// TIA Portal V16 program export: 1 tag tables, 0 data types, 0 data blocks, 6 code blocks (in call order from the OBs), 0 instance data blocks

VAR_GLOBAL   // PLC tag table "Standard-Variablentabelle"
   "Auto/Manual" AT %I0.0 : Bool;
   Start AT %I0.1 : Bool;
   Reset AT %I0.2 : Bool;
   Stop AT %I0.3 : Bool;
   Estop AT %I0.4 : Bool;
   "Conveyor Sensor 1" AT %I0.5 : Bool;
   "Conveyor Sensor 2" AT %I0.6 : Bool;
   "Conveyor Sensor 3" AT %I0.7 : Bool;
   "Alarm Siren" AT %Q0.0 : Bool;
   "Start Light" AT %Q0.1 : Bool;
   "Reset Light" AT %Q0.2 : Bool;
   "Stop Light" AT %Q0.3 : Bool;
   "Pusher 2" AT %Q0.5 : Bool;
   "Stack Light Green" AT %Q0.6 : Bool;
   "Stack Light Yellow" AT %Q0.7 : Bool;
   "Ready to Run" AT %M0.0 : Bool;
   "Reset Memory" AT %M0.5 : Bool;
   "Pusher Sensor 1 Mem" AT %M0.6 : Bool;
   "Pusher 1 FW Mem" AT %M0.7 : Bool;
   "Pusher Sensor 2 Mem" AT %M1.0 : Bool;
   "Pusher 2 FW Mem" AT %M1.1 : Bool;
   "Conveyor Sensor 4" AT %I1.0 : Bool;
   "Pusher Sensor 1" AT %I1.1 : Bool;
   "Pusher Sensor 2" AT %I1.2 : Bool;
   "Pusher 1 FW" AT %I1.3 : Bool;
   "Pusher 2 FW" AT %I1.4 : Bool;
   "Pusher 1" AT %Q0.4 : Bool;
   "Stack Light Red" AT %Q1.0 : Bool;
   "Drain 1" AT %Q1.1 : Bool;
   "Drain 2" AT %Q1.2 : Bool;
   "Drain 3" AT %Q1.3 : Bool;
   "Conveyor 1" AT %QW36 : Int;
   "Conveyor 2" AT %Q1.5 : Bool;
   "Conveyor 3" AT %Q1.6 : Bool;
   "Conveyor 4" AT %Q1.7 : Bool;
   "Conveyor Sensor 1 Mem" AT %M1.2 : Bool;
   "Conveyor Sensor 2 Mem" AT %M1.3 : Bool;
   "Conveyor Sensor 3 Mem" AT %M1.4 : Bool;
   "Conveyor Sensor 4 Mem" AT %M1.5 : Bool;
   "Conveyor Sensor 5 Mem" AT %M1.6 : Bool;
   "Advanced Feeder" AT %Q2.1 : Bool;
   "Conveyor Sensor 5" AT %I1.5 : Bool;
   "Running Torque" AT %IW30 : Int;
   "Running Temperature" AT %IW32 : Int;
   "Error Message" AT %Q2.2 : Bool;
   "1.5 KG" AT %QW30 : Int;
   "5.0 KG" AT %QW32 : Int;
   "7.5" AT %QW34 : Int;
   "Estop Memory" AT %M0.1 : Bool;
END_VAR

ORGANIZATION_BLOCK "Main"   // OB1, LAD, ProgramCycle
TITLE = "Main Program Sweep (Cycle)"
{ S7_Optimized_Access := 'TRUE' }
VERSION : 0.1
// stored: AutoNumber true, IsIECCheckEnabled false, SetENOAutomatically false
   VAR_INPUT
      Initial_Call : Bool;   // Initial call of this OB
      Remanence : Bool;   // =True, if remanent data are available
   END_VAR
BEGIN

REGION Network 1
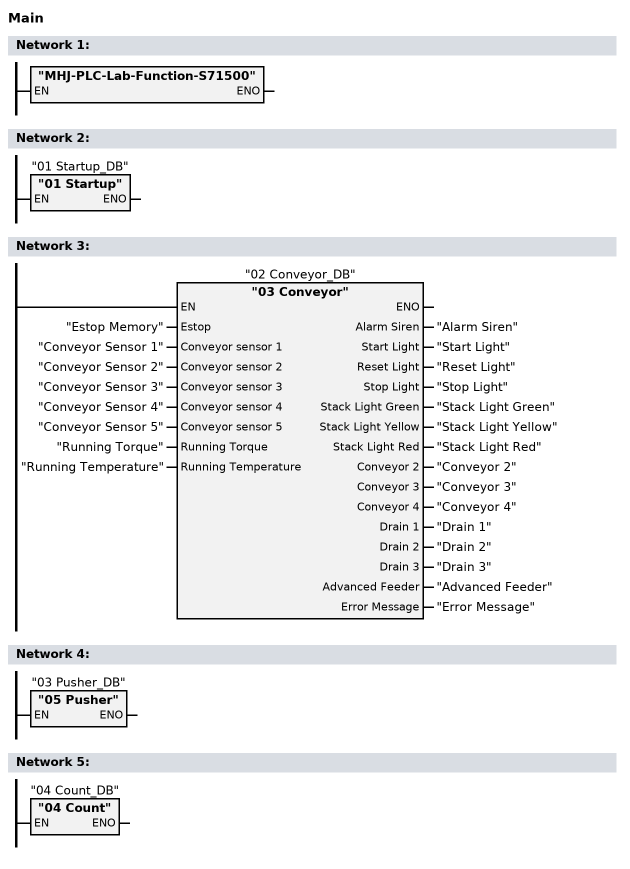
   RUNG wire#powerrail
      "MHJ-PLC-Lab-Function-S71500"()
   END_RUNG
   // the same network as SCL:
   "MHJ-PLC-Lab-Function-S71500"();
END_REGION

REGION Network 2
   RUNG wire#powerrail
      "01 Startup_DB"()
   END_RUNG
   // the same network as SCL:
   "01 Startup_DB"();   // "01 Startup"
END_REGION

REGION Network 3
   RUNG wire#powerrail
      "02 Conveyor_DB"(Estop := "Estop Memory", "Conveyor sensor 1" := "Conveyor Sensor 1", "Conveyor sensor 2" := "Conveyor Sensor 2", "Conveyor sensor 3" := "Conveyor Sensor 3", "Conveyor sensor 4" := "Conveyor Sensor 4", "Conveyor sensor 5" := "Conveyor Sensor 5", "Running Torque" := "Running Torque", "Running Temperature" := "Running Temperature", "Alarm Siren" => "Alarm Siren", "Start Light" => "Start Light", "Reset Light" => "Reset Light", "Stop Light" => "Stop Light", "Stack Light Green" => "Stack Light Green", "Stack Light Yellow" => "Stack Light Yellow", "Stack Light Red" => "Stack Light Red", "Conveyor 2" => "Conveyor 2", "Conveyor 3" => "Conveyor 3", "Conveyor 4" => "Conveyor 4", "Drain 1" => "Drain 1", "Drain 2" => "Drain 2", "Drain 3" => "Drain 3", "Advanced Feeder" => "Advanced Feeder", "Error Message" => "Error Message")
   END_RUNG
   // the same network as SCL:
   "02 Conveyor_DB"(Estop := "Estop Memory",   // "03 Conveyor"
                    "Conveyor sensor 1" := "Conveyor Sensor 1",
                    "Conveyor sensor 2" := "Conveyor Sensor 2",
                    "Conveyor sensor 3" := "Conveyor Sensor 3",
                    "Conveyor sensor 4" := "Conveyor Sensor 4",
                    "Conveyor sensor 5" := "Conveyor Sensor 5",
                    "Running Torque" := "Running Torque",
                    "Running Temperature" := "Running Temperature",
                    "Alarm Siren" => "Alarm Siren",
                    "Start Light" => "Start Light",
                    "Reset Light" => "Reset Light",
                    "Stop Light" => "Stop Light",
                    "Stack Light Green" => "Stack Light Green",
                    "Stack Light Yellow" => "Stack Light Yellow",
                    "Stack Light Red" => "Stack Light Red",
                    "Conveyor 2" => "Conveyor 2",
                    "Conveyor 3" => "Conveyor 3",
                    "Conveyor 4" => "Conveyor 4",
                    "Drain 1" => "Drain 1",
                    "Drain 2" => "Drain 2",
                    "Drain 3" => "Drain 3",
                    "Advanced Feeder" => "Advanced Feeder",
                    "Error Message" => "Error Message");
END_REGION

REGION Network 4
   RUNG wire#powerrail
      "03 Pusher_DB"()
   END_RUNG
   // the same network as SCL:
   "03 Pusher_DB"();   // "05 Pusher"
END_REGION

REGION Network 5
   RUNG wire#powerrail
      "04 Count_DB"()
   END_RUNG
   // the same network as SCL:
   "04 Count_DB"();   // "04 Count"
END_REGION
END_ORGANIZATION_BLOCK

FUNCTION_BLOCK "01 Startup"   // FB1, LAD
{ S7_Optimized_Access := 'TRUE' }
VERSION : 0.1
// stored: AutoNumber true, IsIECCheckEnabled false, IsRetainMemResEnabled false, MemoryReserve 100, SetENOAutomatically false, UDAEnableTagReadback false
   VAR_TEMP   // added for the SCL form of the ladder/FBD networks
      _w1 : Bool;
   END_VAR
BEGIN

REGION Network 1: Run Mode
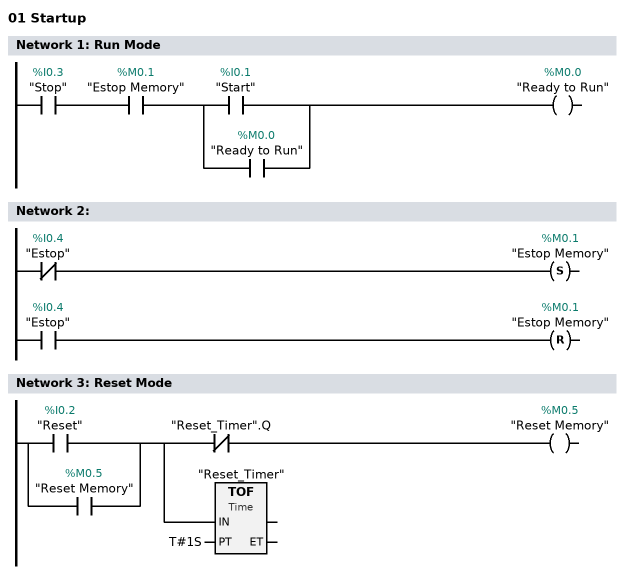
   RUNG wire#powerrail
      Contact( "Stop" )
      Contact( "Estop Memory" )
      wire#w1
      Contact( "Start" )
      wire#w2
      Coil( "Ready to Run" )
   END_RUNG
   RUNG wire#w1
      Contact( "Ready to Run" )
   END_RUNG wire#w2
   // the same network as SCL:
   "Ready to Run" := "Stop" AND "Estop Memory" AND ("Start" OR "Ready to Run");
END_REGION

REGION Network 2
   RUNG wire#powerrail
      I_Contact( "Estop" )
      S_Coil( "Estop Memory" )
   END_RUNG
   RUNG wire#powerrail
      Contact( "Estop" )
      R_Coil( "Estop Memory" )
   END_RUNG
   // the same network as SCL:
   IF NOT "Estop" THEN "Estop Memory" := TRUE; END_IF;
   IF "Estop" THEN "Estop Memory" := FALSE; END_IF;
END_REGION

REGION Network 3: Reset Mode
   RUNG wire#powerrail
      Contact( "Reset" )
      wire#w1
      I_Contact( "Reset_Timer".Q )
      Coil( "Reset Memory" )
   END_RUNG
   RUNG wire#powerrail
      Contact( "Reset Memory" )
   END_RUNG wire#w1
   RUNG wire#w1
      { S7_Templates := "time_type := Time" } "Reset_Timer".TOF(pt := T#1S, et =>)
   END_RUNG
   // the same network as SCL:
   #_w1 := "Reset" OR "Reset Memory";
   "Reset Memory" := #_w1 AND NOT "Reset_Timer".Q;
   "Reset_Timer".TOF(IN := #_w1, PT := T#1S);
END_REGION
END_FUNCTION_BLOCK

FUNCTION_BLOCK "03 Conveyor"
{ S7_Optimized_Access := 'TRUE' }
VERSION : 0.1
   VAR_INPUT 
      Estop : Bool;
      "Conveyor sensor 1" : Bool;
      "Conveyor sensor 2" : Bool;
      "Conveyor sensor 3" : Bool;
      "Conveyor sensor 4" : Bool;
      "Conveyor sensor 5" : Bool;
      "Running Torque" : Int;
      "Running Temperature" : Int;
   END_VAR

   VAR_OUTPUT 
      "Alarm Siren" : Bool;
      "Start Light" : Bool;
      "Reset Light" : Bool;
      "Stop Light" : Bool;
      "Stack Light Green" : Bool;
      "Stack Light Yellow" : Bool;
      "Stack Light Red" : Bool;
      "Conveyor 2" : Bool;
      "Conveyor 3" : Bool;
      "Conveyor 4" : Bool;
      "Drain 1" : Bool;
      "Drain 2" : Bool;
      "Drain 3" : Bool;
      "Advanced Feeder" : Bool;
      "Error Message" : Bool;
   END_VAR

   VAR 
      ET : Time;
      Error : Bool;
   END_VAR


BEGIN
	
	REGION Supply
	    IF "Ready to Run" THEN
	        // Statement section IF
	        #"Advanced Feeder" := TRUE;
	    END_IF;
	    
	    //CONVEYOR 2-5 CONTROL
	    
	    //Conveyor 2
	    IF "Ready to Run" THEN
	        IF #"Conveyor sensor 2" THEN
	            #"Conveyor 2" := TRUE;
	
	            "TOF_2".TOF (IN := #"Conveyor sensor 2",
	            PT := T#30s,
	            Q => #"Conveyor 2",
	            ET => #ET);
	        END_IF
	        ;
	    END_IF;
	    
	    IF "Ready to Run" THEN
	        IF #"Conveyor sensor 3" THEN
	            #"Conveyor 3" := TRUE;
	            
	            "TOF_3".TOF (IN := #"Conveyor sensor 3",
	            PT := T#30s,
	            Q => #"Conveyor 3",
	            ET => #ET);
	            
	        END_IF
	        ;
	    END_IF;
	    
	    IF "Ready to Run" THEN
	        IF #"Conveyor sensor 4" THEN
	            #"Conveyor 4" := TRUE;
	            
	            "TOF_4".TOF (IN := #"Conveyor sensor 4",
	            PT := T#30s,
	            Q => #"Conveyor 4",
	            ET => #ET);
	            
	        END_IF
	        ;
	    END_IF;
	    
	           
	END_REGION
	
	
	REGION Predictive Maintenace
	    
	    IF "Ready to Run" THEN
	        // Statement section IF
	        
	        // IF #"Running Torq > #"Rated Torque"OR #"Running Temperature"> #"Rated Temperature" THEN
	        IF #"Running Torque" > 6 OR #"Running Temperature" > 30 THEN
	            #"Error Message" := TRUE;
	            
	            "Timer_Error".TOF (IN := "Ready to Run",
	            PT := T#300s,
	            Q => #"Error Message",
	            ET => #ET);
	        END_IF;
	    END_IF;
	    
	    IF "Ready to Run" THEN
	        // Statement section IF
	        
	        // IF #"Running Torq > #"Rated Torque"OR #"Running Temperature"> #"Rated Temperature" THEN
	        IF #"Running Torque" > 6 OR #"Running Temperature" > 30 THEN
	            #"Estop" := TRUE;
	            
	            "Timer_Error".TOF(IN := "Ready to Run",
	                              PT := T#600s,
	                              Q => #"Error Message",
	                              ET => #ET);
	        END_IF;
	    END_IF;
	    
	END_REGION
	REGION End
	    IF "Ready to Run" THEN
	        #"Drain 1" := TRUE;
	        #"Drain 2" := TRUE;
	        #"Drain 3" := TRUE;
	    END_IF;
	    
	END_REGION
	
END_FUNCTION_BLOCK

FUNCTION_BLOCK "05 Pusher"   // FB3, LAD
{ S7_Optimized_Access := 'TRUE' }
VERSION : 0.1
// stored: AutoNumber true, IsIECCheckEnabled false, IsRetainMemResEnabled false, MemoryReserve 100, SetENOAutomatically false, UDAEnableTagReadback false
   VAR_TEMP   // added for the SCL form of the ladder/FBD networks
      _w1 : Bool;
      _w2 : Bool;
   END_VAR
BEGIN

REGION Network 1: Sorting by height 1
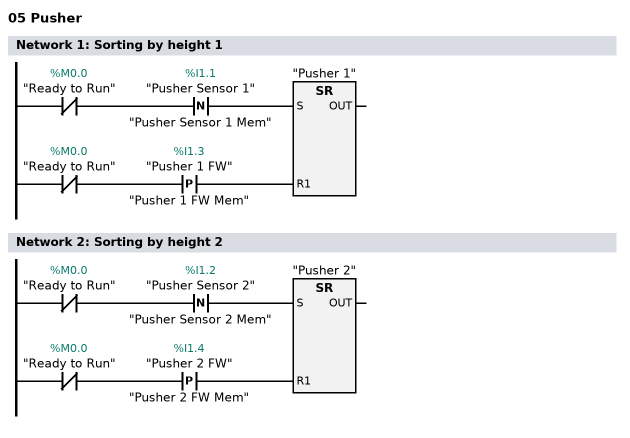
   RUNG wire#powerrail
      I_Contact( "Ready to Run" )
      N_Contact(operand := "Pusher Sensor 1", bit := "Pusher Sensor 1 Mem")
      S_SR(operand := "Pusher 1", r1 := wire#w1)
   END_RUNG
   RUNG wire#powerrail
      I_Contact( "Ready to Run" )
      P_Contact(operand := "Pusher 1 FW", bit := "Pusher 1 FW Mem")
   END_RUNG wire#w1
   // the same network as SCL:
   #_w1 := NOT "Ready to Run" AND NOT "Pusher Sensor 1" AND "Pusher Sensor 1 Mem";   // falling edge of "Pusher Sensor 1"
   "Pusher Sensor 1 Mem" := "Pusher Sensor 1";
   #_w2 := NOT "Ready to Run" AND "Pusher 1 FW" AND NOT "Pusher 1 FW Mem";   // rising edge of "Pusher 1 FW"
   "Pusher 1 FW Mem" := "Pusher 1 FW";
   IF #_w1 THEN
       "Pusher 1" := TRUE;   // SR flip-flop
   END_IF;
   IF #_w2 THEN "Pusher 1" := FALSE; END_IF;
END_REGION

REGION Network 2: Sorting by height 2
   RUNG wire#powerrail
      I_Contact( "Ready to Run" )
      N_Contact(operand := "Pusher Sensor 2", bit := "Pusher Sensor 2 Mem")
      S_SR(operand := "Pusher 2", r1 := wire#w1)
   END_RUNG
   RUNG wire#powerrail
      I_Contact( "Ready to Run" )
      P_Contact(operand := "Pusher 2 FW", bit := "Pusher 2 FW Mem")
   END_RUNG wire#w1
   // the same network as SCL:
   #_w1 := NOT "Ready to Run" AND NOT "Pusher Sensor 2" AND "Pusher Sensor 2 Mem";   // falling edge of "Pusher Sensor 2"
   "Pusher Sensor 2 Mem" := "Pusher Sensor 2";
   #_w2 := NOT "Ready to Run" AND "Pusher 2 FW" AND NOT "Pusher 2 FW Mem";   // rising edge of "Pusher 2 FW"
   "Pusher 2 FW Mem" := "Pusher 2 FW";
   IF #_w1 THEN
       "Pusher 2" := TRUE;   // SR flip-flop
   END_IF;
   IF #_w2 THEN "Pusher 2" := FALSE; END_IF;
END_REGION
END_FUNCTION_BLOCK

FUNCTION_BLOCK "04 Count"   // FB4, LAD
{ S7_Optimized_Access := 'TRUE' }
VERSION : 0.1
// stored: AutoNumber true, IsIECCheckEnabled false, IsRetainMemResEnabled false, MemoryReserve 100, SetENOAutomatically false, UDAEnableTagReadback false
   VAR_TEMP   // added for the SCL form of the ladder/FBD networks
      _w1 : Bool;
      _w2 : Bool;
      _w3 : Bool;
   END_VAR
BEGIN

REGION Network 1: Items count
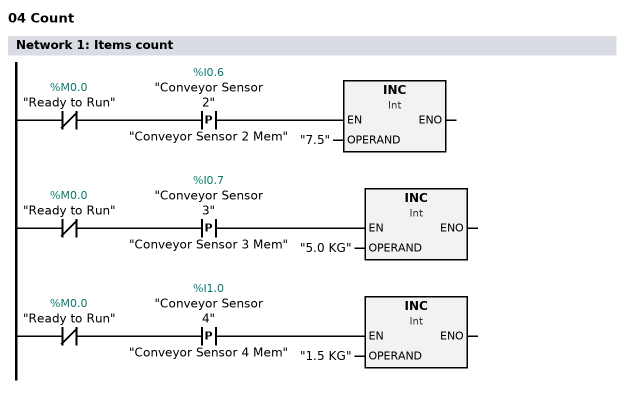
   RUNG wire#powerrail
      I_Contact( "Ready to Run" )
      P_Contact(operand := "Conveyor Sensor 2", bit := "Conveyor Sensor 2 Mem")
      { S7_Templates := "DestType := Int" } Inc( "7.5" )
   END_RUNG
   RUNG wire#powerrail
      I_Contact( "Ready to Run" )
      P_Contact(operand := "Conveyor Sensor 3", bit := "Conveyor Sensor 3 Mem")
      { S7_Templates := "DestType := Int" } Inc( "5.0 KG" )
   END_RUNG
   RUNG wire#powerrail
      I_Contact( "Ready to Run" )
      P_Contact(operand := "Conveyor Sensor 4", bit := "Conveyor Sensor 4 Mem")
      { S7_Templates := "DestType := Int" } Inc( "1.5 KG" )
   END_RUNG
   // the same network as SCL:
   #_w1 := NOT "Ready to Run" AND "Conveyor Sensor 2" AND NOT "Conveyor Sensor 2 Mem";   // rising edge of "Conveyor Sensor 2"
   "Conveyor Sensor 2 Mem" := "Conveyor Sensor 2";
   IF #_w1 THEN "7.5" := "7.5" + 1; END_IF;
   #_w2 := NOT "Ready to Run" AND "Conveyor Sensor 3" AND NOT "Conveyor Sensor 3 Mem";   // rising edge of "Conveyor Sensor 3"
   "Conveyor Sensor 3 Mem" := "Conveyor Sensor 3";
   IF #_w2 THEN "5.0 KG" := "5.0 KG" + 1; END_IF;
   #_w3 := NOT "Ready to Run" AND "Conveyor Sensor 4" AND NOT "Conveyor Sensor 4 Mem";   // rising edge of "Conveyor Sensor 4"
   "Conveyor Sensor 4 Mem" := "Conveyor Sensor 4";
   IF #_w3 THEN "1.5 KG" := "1.5 KG" + 1; END_IF;
END_REGION
END_FUNCTION_BLOCK

FUNCTION_BLOCK "Entry Conveyor"   // FB5, LAD
{ S7_Optimized_Access := 'TRUE' }
VERSION : 0.1
// stored: AutoNumber true, IsIECCheckEnabled false, IsRetainMemResEnabled false, MemoryReserve 100, SetENOAutomatically false, UDAEnableTagReadback false
BEGIN

REGION Network 1
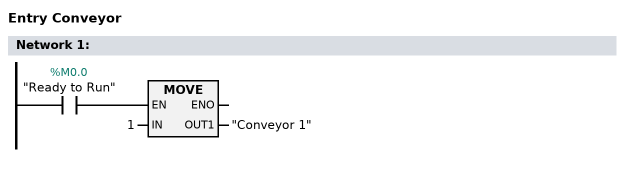
   RUNG wire#powerrail
      Contact( "Ready to Run" )
      Move(in := 1, out1 => "Conveyor 1")
   END_RUNG
   // the same network as SCL:
   IF "Ready to Run" THEN "Conveyor 1" := 1; END_IF;
END_REGION
END_FUNCTION_BLOCK
